FUNCTION_BLOCK TcoSequenceObserverTests EXTENDS TcoCore._internals_TcoContext
VAR				
	_s : TcoCore.TcoSequence(THIS^, eRestoreMode.None);
	_sObserver : TcoCore.TcoSequencerObserver(THIS^);		
END_VAR

(*~
	<docu>
		<summary>
			Main method of the TcoContext. This is the entry point of any control logic that belongs to this context. 
			The call of this method is ensured by calling the <c>InstanceName.Run()</c> method, and it must not be called explicitly.
			This method is abstract, and it must be overridden in derived block.
		</summary>
	</docu>
~*)
METHOD PROTECTED  Main
CASE _testId OF
	eTcoSequenceObserverTests.RestoreSequencer:
		_s.Restore();
		_sObserver.Clear();		
	eTcoSequenceObserverTests.RunSequenceWithObserverTest:
		RunSequencerWithObserver();
	eTcoSequenceObserverTests.RunSequenceWithoutObserverTest:
		RunSequencerWithoutObserver();	
END_CASE
END_METHOD

METHOD RunSequencerWithObserver
VAR_INPUT
END_VAR
_s.Open();

THIS^._s.Observer := _sObserver;

THIS^._s.Messenger.Info('Stations two sequencer is running.');

IF(_s.Step(100, 
		TRUE, 
		'100')) THEN
//-----------------------------------------------------
	_s.StepCompleteWhen(_s.CurrentStep.Duration >= T#10MS);
//-----------------------------------------------------	
END_IF

IF(_s.Step(200, 
		TRUE, 
		'200')) THEN
//-----------------------------------------------------
	_s.StepCompleteWhen(_s.CurrentStep.Duration >= T#20MS);
//-----------------------------------------------------	
END_IF

IF(_s.Step(300, 
		TRUE, 
		'300')) THEN
//-----------------------------------------------------
	_s.StepCompleteWhen(_s.CurrentStep.Duration >= T#30MS);
//-----------------------------------------------------	
END_IF

IF(_s.Step(400, 
		TRUE, 
		'400')) THEN
//-----------------------------------------------------
	_s.StepCompleteWhen(_s.CurrentStep.Duration >= T#40MS);
//-----------------------------------------------------	
END_IF

IF(_s.Step(500, 
		TRUE, 
		'500')) THEN
//-----------------------------------------------------
	THIS^.ProbeDoneWhen(TRUE);
	_s.Restore();
//-----------------------------------------------------	
END_IF

_s.Close();
END_METHOD

METHOD RunSequencerWithoutObserver
VAR_INPUT
END_VAR
_s.Open();

THIS^._s.Observer := 0;

THIS^._s.Messenger.Info('Stations two sequencer is running.');

IF(_s.Step(100, 
		TRUE, 
		'100')) THEN
//-----------------------------------------------------
	_s.StepCompleteWhen(_s.CurrentStep.Duration >= T#250MS);
//-----------------------------------------------------	
END_IF

IF(_s.Step(200, 
		TRUE, 
		'200')) THEN
//-----------------------------------------------------
	_s.StepCompleteWhen(_s.CurrentStep.Duration >= T#100MS);
//-----------------------------------------------------	
END_IF

IF(_s.Step(300, 
		TRUE, 
		'300')) THEN
//-----------------------------------------------------
	_s.StepCompleteWhen(_s.CurrentStep.Duration >= T#50MS);
//-----------------------------------------------------	
END_IF

IF(_s.Step(400, 
		TRUE, 
		'400')) THEN
//-----------------------------------------------------
	_s.StepCompleteWhen(_s.CurrentStep.Duration >= T#25MS);
//-----------------------------------------------------	
END_IF

IF(_s.Step(500, 
		TRUE, 
		'500')) THEN
//-----------------------------------------------------
	THIS^.ProbeDoneWhen(TRUE);
	_s.Restore();
//-----------------------------------------------------	
END_IF

_s.Close();
END_METHOD

END_FUNCTION_BLOCK

(* stored: Version 1.1.0.1
   POU TcoSequenceObserverTests: Id {031e84f0-129a-00ae-272d-2f4b1c1c0910}, SpecialFunc None
   Method Main: Id {cc96ad88-e531-0253-3850-8de33117f9a5}
   Method RunSequencerWithObserver: Id {a0c2b2b1-6da4-0597-1477-816fefac11a2}
   Method RunSequencerWithoutObserver: Id {c8b17968-2047-0c9c-1faa-e93685ccc195} *)
